{attribute addProperty BoxType "AX5201-0000-0011-0011"}
{attribute addProperty Id "Drive_status_wordAT %I*UINT1620Position_feedback_1_valueAT %I*DINT3240"}
{attribute addProperty CRC "43974933"}
{attribute addProperty SizeInBites "48"}
{attribute addProperty SizeInBytes "6"}
TYPE AT_029F0115 :
STRUCT
	{attribute addProperty Name "Drive_status_word"}
	Drive_status_word AT %I* : UINT;
	{attribute addProperty Name "Position_feedback_1_value"}
	Position_feedback_1_value AT %I* : DINT;
END_STRUCT
END_TYPE

(* stored: Version 1.2.0.0, ProductVersion 3.1.4024.9
   DUT AT_029F0115: Id {fc4aa4c0-a074-4409-8cdc-8186675f9de7} *)
